// TIA Portal V20 export
DATA_BLOCK "LPFE_ProgramData"   // DB239
TITLE = LPFE_ProgramData
{ DB_Accessible_From_OPC_UA := 'FALSE' }
AUTHOR : DI FA SUP
FAMILY : LPFE
// Contain the program related data
// stored: Access Published, DBAccessibleFromOPCUA false, DBAccessibleFromWebserver false, MemoryReserve 100, Namespace PFE
   VAR
      PLCInfo : "LPFE_typePLCInfo";   // PLC Information ( Name, Area and Sub Area)
      ProgramInformation : Array[0.._.MAX_NO_PROGRAMS] of "LPFE_typeProgramInfo";   // Array for the information of all programs in the entire PLC .
   END_VAR
BEGIN
   PLCInfo."Name" := 'BA030AZSC1';
   PLCInfo.Area := '';
   PLCInfo.SubArea := '';
   ProgramInformation[0].programName[0] := 'B';
   ProgramInformation[0].programName[1] := 'A';
   ProgramInformation[0].programName[2] := '0';
   ProgramInformation[0].programName[3] := '3';
   ProgramInformation[0].programName[4] := '0';
   ProgramInformation[0].programName[5] := 'A';
   ProgramInformation[0].programName[6] := '_';
   ProgramInformation[0].programName[7] := 'U';
   ProgramInformation[0].programName[8] := '1';
   ProgramInformation[0].programName[9] := 'E';
   ProgramInformation[0].programName[10] := 'm';
   ProgramInformation[0].programName[11..12] := '0';
   ProgramInformation[0].programName[13..15] := '$00';
   ProgramInformation[1].programName[0] := 'B';
   ProgramInformation[1].programName[1] := 'A';
   ProgramInformation[1].programName[2] := '0';
   ProgramInformation[1].programName[3] := '3';
   ProgramInformation[1].programName[4] := '0';
   ProgramInformation[1].programName[5] := 'A';
   ProgramInformation[1].programName[6] := '_';
   ProgramInformation[1].programName[7] := 'U';
   ProgramInformation[1].programName[8] := '1';
   ProgramInformation[1].programName[9] := 'E';
   ProgramInformation[1].programName[10] := 'm';
   ProgramInformation[1].programName[11] := '0';
   ProgramInformation[1].programName[12] := '1';
   ProgramInformation[1].programName[13..15] := '$00';
   ProgramInformation[2].programName[0] := 'B';
   ProgramInformation[2].programName[1] := 'A';
   ProgramInformation[2].programName[2] := '0';
   ProgramInformation[2].programName[3] := '3';
   ProgramInformation[2].programName[4] := '0';
   ProgramInformation[2].programName[5] := 'A';
   ProgramInformation[2].programName[6] := '_';
   ProgramInformation[2].programName[7] := 'U';
   ProgramInformation[2].programName[8] := '1';
   ProgramInformation[2].programName[9] := 'E';
   ProgramInformation[2].programName[10] := 'm';
   ProgramInformation[2].programName[11] := '0';
   ProgramInformation[2].programName[12] := '2';
   ProgramInformation[2].programName[13..15] := '$00';
   ProgramInformation[3].programName[0] := 'B';
   ProgramInformation[3].programName[1] := 'A';
   ProgramInformation[3].programName[2] := '0';
   ProgramInformation[3].programName[3] := '3';
   ProgramInformation[3].programName[4] := '0';
   ProgramInformation[3].programName[5] := 'A';
   ProgramInformation[3].programName[6] := '_';
   ProgramInformation[3].programName[7] := 'U';
   ProgramInformation[3].programName[8] := '1';
   ProgramInformation[3].programName[9] := 'E';
   ProgramInformation[3].programName[10] := 'm';
   ProgramInformation[3].programName[11] := '0';
   ProgramInformation[3].programName[12] := '3';
   ProgramInformation[3].programName[13..15] := '$00';
   ProgramInformation[4].programName[0] := 'B';
   ProgramInformation[4].programName[1] := 'A';
   ProgramInformation[4].programName[2] := '0';
   ProgramInformation[4].programName[3] := '3';
   ProgramInformation[4].programName[4] := '0';
   ProgramInformation[4].programName[5] := 'A';
   ProgramInformation[4].programName[6] := '_';
   ProgramInformation[4].programName[7] := 'U';
   ProgramInformation[4].programName[8] := '1';
   ProgramInformation[4].programName[9] := 'E';
   ProgramInformation[4].programName[10] := 'm';
   ProgramInformation[4].programName[11] := '0';
   ProgramInformation[4].programName[12] := '4';
   ProgramInformation[4].programName[13..15] := '$00';
   ProgramInformation[5].programName[0] := 'B';
   ProgramInformation[5].programName[1] := 'A';
   ProgramInformation[5].programName[2] := '0';
   ProgramInformation[5].programName[3] := '3';
   ProgramInformation[5].programName[4] := '0';
   ProgramInformation[5].programName[5] := 'A';
   ProgramInformation[5].programName[6] := '_';
   ProgramInformation[5].programName[7] := 'U';
   ProgramInformation[5].programName[8] := '1';
   ProgramInformation[5].programName[9] := 'E';
   ProgramInformation[5].programName[10] := 'm';
   ProgramInformation[5].programName[11] := '0';
   ProgramInformation[5].programName[12] := '5';
   ProgramInformation[5].programName[13..15] := '$00';
   ProgramInformation[6].programName[0] := 'B';
   ProgramInformation[6].programName[1] := 'A';
   ProgramInformation[6].programName[2] := '0';
   ProgramInformation[6].programName[3] := '3';
   ProgramInformation[6].programName[4] := '0';
   ProgramInformation[6].programName[5] := 'A';
   ProgramInformation[6].programName[6] := '_';
   ProgramInformation[6].programName[7] := 'U';
   ProgramInformation[6].programName[8] := '1';
   ProgramInformation[6].programName[9] := 'E';
   ProgramInformation[6].programName[10] := 'm';
   ProgramInformation[6].programName[11] := '0';
   ProgramInformation[6].programName[12] := '6';
   ProgramInformation[6].programName[13..15] := '$00';
   ProgramInformation[7].programName[0] := 'B';
   ProgramInformation[7].programName[1] := 'A';
   ProgramInformation[7].programName[2] := '0';
   ProgramInformation[7].programName[3] := '3';
   ProgramInformation[7].programName[4] := '0';
   ProgramInformation[7].programName[5] := 'A';
   ProgramInformation[7].programName[6] := '_';
   ProgramInformation[7].programName[7] := 'U';
   ProgramInformation[7].programName[8] := '1';
   ProgramInformation[7].programName[9] := 'E';
   ProgramInformation[7].programName[10] := 'm';
   ProgramInformation[7].programName[11] := '0';
   ProgramInformation[7].programName[12] := '7';
   ProgramInformation[7].programName[13..15] := '$00';
   ProgramInformation[8].programName[0] := 'B';
   ProgramInformation[8].programName[1] := 'A';
   ProgramInformation[8].programName[2] := '0';
   ProgramInformation[8].programName[3] := '3';
   ProgramInformation[8].programName[4] := '0';
   ProgramInformation[8].programName[5] := 'A';
   ProgramInformation[8].programName[6] := '_';
   ProgramInformation[8].programName[7] := 'U';
   ProgramInformation[8].programName[8] := '1';
   ProgramInformation[8].programName[9] := 'E';
   ProgramInformation[8].programName[10] := 'm';
   ProgramInformation[8].programName[11] := '0';
   ProgramInformation[8].programName[12] := '8';
   ProgramInformation[8].programName[13..15] := '$00';
   ProgramInformation[9].programName[0] := 'B';
   ProgramInformation[9].programName[1] := 'A';
   ProgramInformation[9].programName[2] := '0';
   ProgramInformation[9].programName[3] := '3';
   ProgramInformation[9].programName[4] := '0';
   ProgramInformation[9].programName[5] := 'A';
   ProgramInformation[9].programName[6] := '_';
   ProgramInformation[9].programName[7] := 'U';
   ProgramInformation[9].programName[8] := '1';
   ProgramInformation[9].programName[9] := 'E';
   ProgramInformation[9].programName[10] := 'm';
   ProgramInformation[9].programName[11] := '0';
   ProgramInformation[9].programName[12] := '9';
   ProgramInformation[9].programName[13..15] := '$00';
   ProgramInformation[10].programName[0] := 'B';
   ProgramInformation[10].programName[1] := 'A';
   ProgramInformation[10].programName[2] := '0';
   ProgramInformation[10].programName[3] := '3';
   ProgramInformation[10].programName[4] := '0';
   ProgramInformation[10].programName[5] := 'A';
   ProgramInformation[10].programName[6] := '_';
   ProgramInformation[10].programName[7] := 'U';
   ProgramInformation[10].programName[8] := '1';
   ProgramInformation[10].programName[9] := 'E';
   ProgramInformation[10].programName[10] := 'm';
   ProgramInformation[10].programName[11] := '1';
   ProgramInformation[10].programName[12] := '0';
   ProgramInformation[10].programName[13..15] := '$00';
   ProgramInformation[11].programName[0] := 'B';
   ProgramInformation[11].programName[1] := 'A';
   ProgramInformation[11].programName[2] := '0';
   ProgramInformation[11].programName[3] := '3';
   ProgramInformation[11].programName[4] := '0';
   ProgramInformation[11].programName[5] := 'A';
   ProgramInformation[11].programName[6] := '_';
   ProgramInformation[11].programName[7] := 'U';
   ProgramInformation[11].programName[8] := '1';
   ProgramInformation[11].programName[9] := 'E';
   ProgramInformation[11].programName[10] := 'm';
   ProgramInformation[11].programName[11..12] := '1';
   ProgramInformation[11].programName[13..15] := '$00';
   ProgramInformation[12].programName[0] := 'B';
   ProgramInformation[12].programName[1] := 'A';
   ProgramInformation[12].programName[2] := '0';
   ProgramInformation[12].programName[3] := '3';
   ProgramInformation[12].programName[4] := '0';
   ProgramInformation[12].programName[5] := 'A';
   ProgramInformation[12].programName[6] := '_';
   ProgramInformation[12].programName[7] := 'U';
   ProgramInformation[12].programName[8] := '1';
   ProgramInformation[12].programName[9] := 'E';
   ProgramInformation[12].programName[10] := 'm';
   ProgramInformation[12].programName[11] := '1';
   ProgramInformation[12].programName[12] := '2';
   ProgramInformation[12].programName[13..15] := '$00';
   ProgramInformation[13].programName[0] := 'B';
   ProgramInformation[13].programName[1] := 'A';
   ProgramInformation[13].programName[2] := '0';
   ProgramInformation[13].programName[3] := '3';
   ProgramInformation[13].programName[4] := '0';
   ProgramInformation[13].programName[5] := 'A';
   ProgramInformation[13].programName[6] := '_';
   ProgramInformation[13].programName[7] := 'U';
   ProgramInformation[13].programName[8] := '1';
   ProgramInformation[13].programName[9] := 'E';
   ProgramInformation[13].programName[10] := 'm';
   ProgramInformation[13].programName[11] := '1';
   ProgramInformation[13].programName[12] := '3';
   ProgramInformation[13].programName[13..15] := '$00';
   ProgramInformation[14].programName[0] := 'B';
   ProgramInformation[14].programName[1] := 'A';
   ProgramInformation[14].programName[2] := '0';
   ProgramInformation[14].programName[3] := '3';
   ProgramInformation[14].programName[4] := '0';
   ProgramInformation[14].programName[5] := 'A';
   ProgramInformation[14].programName[6] := '_';
   ProgramInformation[14].programName[7] := 'U';
   ProgramInformation[14].programName[8] := '1';
   ProgramInformation[14].programName[9] := 'E';
   ProgramInformation[14].programName[10] := 'm';
   ProgramInformation[14].programName[11] := '1';
   ProgramInformation[14].programName[12] := '4';
   ProgramInformation[14].programName[13..15] := '$00';
   ProgramInformation[15].programName[0] := 'B';
   ProgramInformation[15].programName[1] := 'A';
   ProgramInformation[15].programName[2] := '0';
   ProgramInformation[15].programName[3] := '3';
   ProgramInformation[15].programName[4] := '0';
   ProgramInformation[15].programName[5] := 'A';
   ProgramInformation[15].programName[6] := '_';
   ProgramInformation[15].programName[7] := 'U';
   ProgramInformation[15].programName[8] := '1';
   ProgramInformation[15].programName[9] := 'E';
   ProgramInformation[15].programName[10] := 'm';
   ProgramInformation[15].programName[11] := '1';
   ProgramInformation[15].programName[12] := '5';
   ProgramInformation[15].programName[13..15] := '$00';
   ProgramInformation[16].programName[0] := 'B';
   ProgramInformation[16].programName[1] := 'A';
   ProgramInformation[16].programName[2] := '0';
   ProgramInformation[16].programName[3] := '3';
   ProgramInformation[16].programName[4] := '0';
   ProgramInformation[16].programName[5] := 'A';
   ProgramInformation[16].programName[6] := '_';
   ProgramInformation[16].programName[7] := 'U';
   ProgramInformation[16].programName[8] := '1';
   ProgramInformation[16].programName[9] := 'E';
   ProgramInformation[16].programName[10] := 'm';
   ProgramInformation[16].programName[11] := '1';
   ProgramInformation[16].programName[12] := '6';
   ProgramInformation[16].programName[13..15] := '$00';
   ProgramInformation[17].programName[0] := 'B';
   ProgramInformation[17].programName[1] := 'A';
   ProgramInformation[17].programName[2] := '0';
   ProgramInformation[17].programName[3] := '3';
   ProgramInformation[17].programName[4] := '0';
   ProgramInformation[17].programName[5] := 'A';
   ProgramInformation[17].programName[6] := '_';
   ProgramInformation[17].programName[7] := 'U';
   ProgramInformation[17].programName[8] := '1';
   ProgramInformation[17].programName[9] := 'E';
   ProgramInformation[17].programName[10] := 'm';
   ProgramInformation[17].programName[11] := '1';
   ProgramInformation[17].programName[12] := '7';
   ProgramInformation[17].programName[13..15] := '$00';
   ProgramInformation[18].programName[0] := 'B';
   ProgramInformation[18].programName[1] := 'A';
   ProgramInformation[18].programName[2] := '0';
   ProgramInformation[18].programName[3] := '3';
   ProgramInformation[18].programName[4] := '0';
   ProgramInformation[18].programName[5] := 'A';
   ProgramInformation[18].programName[6] := '_';
   ProgramInformation[18].programName[7] := 'U';
   ProgramInformation[18].programName[8] := '1';
   ProgramInformation[18].programName[9] := 'E';
   ProgramInformation[18].programName[10] := 'm';
   ProgramInformation[18].programName[11] := '1';
   ProgramInformation[18].programName[12] := '8';
   ProgramInformation[18].programName[13..15] := '$00';
   ProgramInformation[19].programName[0] := 'B';
   ProgramInformation[19].programName[1] := 'A';
   ProgramInformation[19].programName[2] := '0';
   ProgramInformation[19].programName[3] := '3';
   ProgramInformation[19].programName[4] := '0';
   ProgramInformation[19].programName[5] := 'A';
   ProgramInformation[19].programName[6] := '_';
   ProgramInformation[19].programName[7] := 'U';
   ProgramInformation[19].programName[8] := '1';
   ProgramInformation[19].programName[9] := 'E';
   ProgramInformation[19].programName[10] := 'm';
   ProgramInformation[19].programName[11] := '1';
   ProgramInformation[19].programName[12] := '9';
   ProgramInformation[19].programName[13..15] := '$00';
   ProgramInformation[20].programName[0] := 'B';
   ProgramInformation[20].programName[1] := 'A';
   ProgramInformation[20].programName[2] := '0';
   ProgramInformation[20].programName[3] := '3';
   ProgramInformation[20].programName[4] := '0';
   ProgramInformation[20].programName[5] := 'A';
   ProgramInformation[20].programName[6] := '_';
   ProgramInformation[20].programName[7] := 'U';
   ProgramInformation[20].programName[8] := '1';
   ProgramInformation[20].programName[9] := 'E';
   ProgramInformation[20].programName[10] := 'm';
   ProgramInformation[20].programName[11] := '2';
   ProgramInformation[20].programName[12] := '0';
   ProgramInformation[20].programName[13..15] := '$00';
   ProgramInformation[0].plcOffset := 5000;
   ProgramInformation[1].plcOffset := 5001;
   ProgramInformation[2].plcOffset := 5002;
   ProgramInformation[3].plcOffset := 5003;
   ProgramInformation[4].plcOffset := 5004;
   ProgramInformation[5].plcOffset := 5005;
   ProgramInformation[6].plcOffset := 5006;
   ProgramInformation[7].plcOffset := 5007;
   ProgramInformation[8].plcOffset := 5008;
   ProgramInformation[9].plcOffset := 5009;
   ProgramInformation[10].plcOffset := 5010;
   ProgramInformation[11].plcOffset := 5011;
   ProgramInformation[12].plcOffset := 5012;
   ProgramInformation[13].plcOffset := 5013;
   ProgramInformation[14].plcOffset := 5014;
   ProgramInformation[15].plcOffset := 5015;
   ProgramInformation[16].plcOffset := 5016;
   ProgramInformation[17].plcOffset := 5017;
   ProgramInformation[18].plcOffset := 5018;
   ProgramInformation[19].plcOffset := 5019;
   ProgramInformation[20].plcOffset := 5020;
END_DATA_BLOCK
